ABB RobotStudio station: Step_suction_gripper_20200824-203241.rsstn

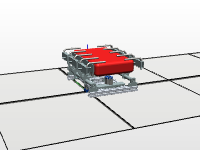
Station Step_suction_gripper (saved by RobotStudio 6.8.8307.1040)
Layout (positions relative to the parent item):
  - T_GRIPPER_2 [graphiccomponentgroup] at (-345.02, -333, 492.44) mm, rotated rx 180 ry 0 rz 0 deg
    - 1046 [graphiccomponentgroup] at (435.5, 105.5, 314.43) mm, rotated rx -90 ry 0 rz 180 deg
      - 1036 [part] at (225.5, -1596.5, -697) mm, rotated rx 0 ry -90 rz -90 deg
      - 1037 [part] at (22.5, 21, 5.41) mm, rotated rx -90 ry 0 rz -90 deg
      - 1038 [part] at (697, -1596.5, 180.5) mm, rotated rx 90 ry 0 rz 180 deg
      - 1039 [part] at (-5.41, 21, -22.5) mm, rotated rx 0 ry 0 rz -90 deg
      - 2.2.001.10.4545.01_kose baglanti duz 45x45_step_MODEL [part]
    - 1048 [graphiccomponentgroup] at (255.5, -60, 272.43) mm, rotated rx 90 ry 0 rz 0 deg
      - 1036 [part] at (225.5, -1596.5, -697) mm, rotated rx 0 ry -90 rz -90 deg
      - 1037 [part] at (22.5, 21, 5.41) mm, rotated rx -90 ry 0 rz -90 deg
      - 1038 [part] at (697, -1596.5, 180.5) mm, rotated rx 90 ry 0 rz 180 deg
      - 1039 [part] at (-5.41, 21, -22.5) mm, rotated rx 0 ry 0 rz -90 deg
      - 2.2.001.10.4545.01_kose baglanti duz 45x45_step_MODEL [part]
    - 1049 [graphiccomponentgroup] at (435.5, 60.5, 272.43) mm, rotated rx 90 ry 0 rz 180 deg
      - 1036 [part] at (225.5, -1596.5, -697) mm, rotated rx 0 ry -90 rz -90 deg
      - 1037 [part] at (22.5, 21, 5.41) mm, rotated rx -90 ry 0 rz -90 deg
      - 1038 [part] at (697, -1596.5, 180.5) mm, rotated rx 90 ry 0 rz 180 deg
      - 1039 [part] at (-5.41, 21, -22.5) mm, rotated rx 0 ry 0 rz -90 deg
      - 2.2.001.10.4545.01_kose baglanti duz 45x45_step_MODEL [part]
    - 1050 [graphiccomponentgroup] at (255.5, 60.5, 314.43) mm, rotated rx -90 ry 0 rz 0 deg
      - 1036 [part] at (225.5, -1596.5, -697) mm, rotated rx 0 ry -90 rz -90 deg
      - 1037 [part] at (22.5, 21, 5.41) mm, rotated rx -90 ry 0 rz -90 deg
      - 1038 [part] at (697, -1596.5, 180.5) mm, rotated rx 90 ry 0 rz 180 deg
      - 1039 [part] at (-5.41, 21, -22.5) mm, rotated rx 0 ry 0 rz -90 deg
      - 2.2.001.10.4545.01_kose baglanti duz 45x45_step_MODEL [part]
    - 1051 [graphiccomponentgroup] at (255, 255, 272.43) mm, rotated rx 90 ry 0 rz -90 deg
      - 1036 [part] at (225.5, -1596.5, -697) mm, rotated rx 0 ry -90 rz -90 deg
      - 1037 [part] at (22.5, 21, 5.41) mm, rotated rx -90 ry 0 rz -90 deg
      - 1038 [part] at (697, -1596.5, 180.5) mm, rotated rx 90 ry 0 rz 180 deg
      - 1039 [part] at (-5.41, 21, -22.5) mm, rotated rx 0 ry 0 rz -90 deg
      - 2.2.001.10.4545.01_kose baglanti duz 45x45_step_MODEL [part]
    - 1052 [graphiccomponentgroup] at (480, -255, 314.43) mm, rotated rx -90 ry 0 rz 90 deg
      - 1036 [part] at (225.5, -1596.5, -697) mm, rotated rx 0 ry -90 rz -90 deg
      - 1037 [part] at (22.5, 21, 5.41) mm, rotated rx -90 ry 0 rz -90 deg
      - 1038 [part] at (697, -1596.5, 180.5) mm, rotated rx 90 ry 0 rz 180 deg
      - 1039 [part] at (-5.41, 21, -22.5) mm, rotated rx 0 ry 0 rz -90 deg
      - 2.2.001.10.4545.01_kose baglanti duz 45x45_step_MODEL [part]
    - 1055 [graphiccomponentgroup] at (255.5, -105, 314.43) mm, rotated rx -90 ry 0 rz 0 deg
      - 1036 [part] at (225.5, -1596.5, -697) mm, rotated rx 0 ry -90 rz -90 deg
      - 1037 [part] at (22.5, 21, 5.41) mm, rotated rx -90 ry 0 rz -90 deg
      - 1038 [part] at (697, -1596.5, 180.5) mm, rotated rx 90 ry 0 rz 180 deg
      - 1039 [part] at (-5.41, 21, -22.5) mm, rotated rx 0 ry 0 rz -90 deg
      - 2.2.001.10.4545.01_kose baglanti duz 45x45_step_MODEL [part]
    - 1059 [graphiccomponentgroup] at (435.5, -105, 272.43) mm, rotated rx 90 ry 0 rz 180 deg
      - 1036 [part] at (225.5, -1596.5, -697) mm, rotated rx 0 ry -90 rz -90 deg
      - 1037 [part] at (22.5, 21, 5.41) mm, rotated rx -90 ry 0 rz -90 deg
      - 1038 [part] at (697, -1596.5, 180.5) mm, rotated rx 90 ry 0 rz 180 deg
      - 1039 [part] at (-5.41, 21, -22.5) mm, rotated rx 0 ry 0 rz -90 deg
      - 2.2.001.10.4545.01_kose baglanti duz 45x45_step_MODEL [part]
    - 1061 [graphiccomponentgroup] at (435, 255, 314.43) mm, rotated rx -90 ry 0 rz -90 deg
      - 1036 [part] at (225.5, -1596.5, -697) mm, rotated rx 0 ry -90 rz -90 deg
      - 1037 [part] at (22.5, 21, 5.41) mm, rotated rx -90 ry 0 rz -90 deg
      - 1038 [part] at (697, -1596.5, 180.5) mm, rotated rx 90 ry 0 rz 180 deg
      - 1039 [part] at (-5.41, 21, -22.5) mm, rotated rx 0 ry 0 rz -90 deg
      - 2.2.001.10.4545.01_kose baglanti duz 45x45_step_MODEL [part]
    - 1062 [graphiccomponentgroup] at (255, -255, 314.43) mm, rotated rx -90 ry 0 rz 90 deg
      - 1036 [part] at (225.5, -1596.5, -697) mm, rotated rx 0 ry -90 rz -90 deg
      - 1037 [part] at (22.5, 21, 5.41) mm, rotated rx -90 ry 0 rz -90 deg
      - 1038 [part] at (697, -1596.5, 180.5) mm, rotated rx 90 ry 0 rz 180 deg
      - 1039 [part] at (-5.41, 21, -22.5) mm, rotated rx 0 ry 0 rz -90 deg
      - 2.2.001.10.4545.01_kose baglanti duz 45x45_step_MODEL [part]
    - 1063 [graphiccomponentgroup] at (537.5, 287.5, 249.93) mm, rotated rx 180 ry 0 rz -90 deg
      - 1035 [graphiccomponentgroup] at (5, 0, 30) mm
        - 1032 [part]
        - 1033 [part]
        - 1034 [part]
      - RULMAN_YATAK [part]
    - 1064 [graphiccomponentgroup] at (435.5, -60, 314.43) mm, rotated rx -90 ry 0 rz 180 deg
      - 1036 [part] at (225.5, -1596.5, -697) mm, rotated rx 0 ry -90 rz -90 deg
      - 1037 [part] at (22.5, 21, 5.41) mm, rotated rx -90 ry 0 rz -90 deg
      - 1038 [part] at (697, -1596.5, 180.5) mm, rotated rx 90 ry 0 rz 180 deg
      - 1039 [part] at (-5.41, 21, -22.5) mm, rotated rx 0 ry 0 rz -90 deg
      - 2.2.001.10.4545.01_kose baglanti duz 45x45_step_MODEL [part]
    - 1065 [graphiccomponentgroup] at (210, 255, 314.43) mm, rotated rx -90 ry 0 rz -90 deg
      - 1036 [part] at (225.5, -1596.5, -697) mm, rotated rx 0 ry -90 rz -90 deg
      - 1037 [part] at (22.5, 21, 5.41) mm, rotated rx -90 ry 0 rz -90 deg
      - 1038 [part] at (697, -1596.5, 180.5) mm, rotated rx 90 ry 0 rz 180 deg
      - 1039 [part] at (-5.41, 21, -22.5) mm, rotated rx 0 ry 0 rz -90 deg
      - 2.2.001.10.4545.01_kose baglanti duz 45x45_step_MODEL [part]
    - 1066 [graphiccomponentgroup] at (255.5, 105.5, 272.43) mm, rotated rx 90 ry 0 rz 0 deg
      - 1036 [part] at (225.5, -1596.5, -697) mm, rotated rx 0 ry -90 rz -90 deg
      - 1037 [part] at (22.5, 21, 5.41) mm, rotated rx -90 ry 0 rz -90 deg
      - 1038 [part] at (697, -1596.5, 180.5) mm, rotated rx 90 ry 0 rz 180 deg
      - 1039 [part] at (-5.41, 21, -22.5) mm, rotated rx 0 ry 0 rz -90 deg
      - 2.2.001.10.4545.01_kose baglanti duz 45x45_step_MODEL [part]
    - 1067 [graphiccomponentgroup] at (152.5, -287.5, 249.93) mm, rotated rx 180 ry 0 rz 90 deg
      - 1035 [graphiccomponentgroup] at (5, 0, 30) mm
        - 1032 [part]
        - 1033 [part]
        - 1034 [part]
      - RULMAN_YATAK [part]
    - 1070 [graphiccomponentgroup] at (538.22, -287.5, 251.07) mm, rotated rx 180 ry 0 rz 90 deg
      - 1035 [graphiccomponentgroup] at (5, 0, 30) mm
        - 1032 [part]
        - 1033 [part]
        - 1034 [part]
      - RULMAN_YATAK [part]
    - 1071 [graphiccomponentgroup] at (152.5, 287.5, 249.93) mm, rotated rx 180 ry 0 rz -90 deg
      - 1035 [graphiccomponentgroup] at (5, 0, 30) mm
        - 1032 [part]
        - 1033 [part]
        - 1034 [part]
      - RULMAN_YATAK [part]
    - 1072 [graphiccomponentgroup] at (435, -255, 272.43) mm, rotated rx 90 ry 0 rz 90 deg
      - 1036 [part] at (225.5, -1596.5, -697) mm, rotated rx 0 ry -90 rz -90 deg
      - 1037 [part] at (22.5, 21, 5.41) mm, rotated rx -90 ry 0 rz -90 deg
      - 1038 [part] at (697, -1596.5, 180.5) mm, rotated rx 90 ry 0 rz 180 deg
      - 1039 [part] at (-5.41, 21, -22.5) mm, rotated rx 0 ry 0 rz -90 deg
      - 2.2.001.10.4545.01_kose baglanti duz 45x45_step_MODEL [part]
    - 1073 [graphiccomponentgroup] at (480, 255, 272.43) mm, rotated rx 90 ry 0 rz -90 deg
      - 1036 [part] at (225.5, -1596.5, -697) mm, rotated rx 0 ry -90 rz -90 deg
      - 1037 [part] at (22.5, 21, 5.41) mm, rotated rx -90 ry 0 rz -90 deg
      - 1038 [part] at (697, -1596.5, 180.5) mm, rotated rx 90 ry 0 rz 180 deg
      - 1039 [part] at (-5.41, 21, -22.5) mm, rotated rx 0 ry 0 rz -90 deg
      - 2.2.001.10.4545.01_kose baglanti duz 45x45_step_MODEL [part]
    - 1075 [graphiccomponentgroup] at (210, -255, 272.43) mm, rotated rx 90 ry 0 rz 90 deg
      - 1036 [part] at (225.5, -1596.5, -697) mm, rotated rx 0 ry -90 rz -90 deg
      - 1037 [part] at (22.5, 21, 5.41) mm, rotated rx -90 ry 0 rz -90 deg
      - 1038 [part] at (697, -1596.5, 180.5) mm, rotated rx 90 ry 0 rz 180 deg
      - 1039 [part] at (-5.41, 21, -22.5) mm, rotated rx 0 ry 0 rz -90 deg
      - 2.2.001.10.4545.01_kose baglanti duz 45x45_step_MODEL [part]
    - 1076 [graphiccomponentgroup] at (152.5, -244, 219.93) mm, rotated rx -1.14 ry 0 rz 90 deg
      - 1021 [graphiccomponentgroup] at (505.5, 0, 0) mm, rotated rx 180 ry 0 rz 180 deg
        - 1005 [part] at (523, 0, 0) mm, rotated rx 0 ry 0 rz -90 deg
        - 1006 [part] at (0, 0, 0) mm, rotated rx 0 ry 0 rz 90 deg
        - GR1_P1-2 [part]
      - 1022 [graphiccomponentgroup] at (244, -1, -144) mm, rotated rx 0 ry 90 rz -90 deg
        - 1007 [part] at (0, 215, 0.5) mm, rotated rx -90 ry 0 rz 180 deg
        - 1008 [part] at (0, -35, 0.5) mm, rotated rx -90 ry 0 rz 180 deg
        - 1009 [part] at (0, -215, 0.5) mm, rotated rx -90 ry 0 rz 180 deg
        - GR1_P4 [part]
      - 1023 [part] at (371.5, 54.54, -79.76) mm, rotated rx 0 ry 0.38 rz -90 deg
      - 1024 [part] at (394, 68.87, -207.14) mm, rotated rx 0 ry 0.38 rz -90 deg
      - 1025 [part] at (244, 68.47, -146.98) mm, rotated rx 0.38 ry 0 rz 0 deg
      - 1026 [part] at (94, 68.87, -207.14) mm, rotated rx 0 ry 0.38 rz -90 deg
      - 1027 [part] at (-56, 68.87, -207.14) mm, rotated rx 0 ry 0.38 rz -90 deg
      - 1028 [part] at (244, 68.87, -207.14) mm, rotated rx 0 ry 0.38 rz -90 deg
      - 1029 [part] at (124.5, 54.54, -79.76) mm, rotated rx 0 ry 0.38 rz -90 deg
      - 1030 [part] at (544, 68.87, -207.14) mm, rotated rx 0 ry 0.38 rz -90 deg
      - 1031 [part] at (-94, 0, 0) mm, rotated rx 0 ry 30.38 rz 90 deg
    - 1077 [graphiccomponentgroup] at (538.22, 244, 221.07) mm, rotated rx -0.38 ry 0 rz -90 deg
      - 1010 [graphiccomponentgroup] at (-17.5, 0, 0) mm
        - 1005 [part] at (523, 0, 0) mm, rotated rx 0 ry 0 rz -90 deg
        - 1006 [part] at (0, 0, 0) mm, rotated rx 0 ry 0 rz 90 deg
        - GR1_P1-2 [part]
      - 1011 [graphiccomponentgroup] at (244, -1, -144) mm, rotated rx 0 ry 90 rz -90 deg
        - 1007 [part] at (0, 215, 0.5) mm, rotated rx -90 ry 0 rz 180 deg
        - 1008 [part] at (0, -35, 0.5) mm, rotated rx -90 ry 0 rz 180 deg
        - 1009 [part] at (0, -215, 0.5) mm, rotated rx -90 ry 0 rz 180 deg
        - GR1_P4 [part]
      - 1012 [part] at (371.5, 54.54, -79.76) mm, rotated rx 0 ry 0.38 rz -90 deg
      - 1013 [part] at (394, 68.87, -207.14) mm, rotated rx 0 ry 0.38 rz -90 deg
      - 1014 [part] at (244, 68.47, -146.98) mm, rotated rx 0.38 ry 0 rz 0 deg
      - 1015 [part] at (94, 68.87, -207.14) mm, rotated rx 0 ry 0.38 rz -90 deg
      - 1016 [part] at (-56, 68.87, -207.14) mm, rotated rx 0 ry 0.38 rz -90 deg
      - 1017 [part] at (244, 68.87, -207.14) mm, rotated rx 0 ry 0.38 rz -90 deg
      - 1018 [part] at (124.5, 54.54, -79.76) mm, rotated rx 0 ry 0.38 rz -90 deg
      - 1019 [part] at (544, 68.87, -207.14) mm, rotated rx 0 ry 0.38 rz -90 deg
      - 1020 [part] at (572, 0, 0) mm, rotated rx 0 ry 30.38 rz 90 deg
    - 1079 [graphiccomponentgroup] at (345.02, -333, 408.94) mm, rotated rx 180 ry 0 rz 180 deg
      - 1003 [part]
      - 1004 [part]
    - 1084 [graphiccomponentgroup] at (345, -179.5, 242.67) mm, rotated rx 180 ry 0 rz 90 deg
      - 1001 [part] at (0, 0, 33) mm
      - 1002 [part]
    - 1085 [graphiccomponentgroup] at (345, 179.5, 242.67) mm, rotated rx 180 ry 0 rz -90 deg
      - 1001 [part] at (0, 0, 33) mm
      - 1002 [part]
    - 1047 [part] at (375, -82.5, 294.93) mm, rotated rx 0 ry -90 rz -180 deg
    - 1053 [part] at (375, 82.5, 294.93) mm, rotated rx 0 ry -90 rz -180 deg
    - 1054 [part] at (-110, 277.5, 294.93) mm, rotated rx 0 ry -90 rz -180 deg
    - CAJA [part] at (-1373.11, 0, 0) mm
    - 1057 [part] at (345, -2.5, 317.43) mm
    - 1058 [part] at (-110, -277.5, 294.93) mm, rotated rx 0 ry -90 rz -180 deg
    - 1060 [part] at (232.5, -480, 294.93) mm, rotated rx 0 ry -90 rz -90 deg
    - 1069 [part] at (457.5, -480, 294.93) mm, rotated rx 0 ry -90 rz -90 deg
    - 1078 [part] at (265.02, -345.5, 237.16) mm, rotated rx 0 ry 0 rz 90 deg
    - 1080 [part] at (345.02, -300, 317.44) mm, rotated rx 0 ry 0 rz 90 deg
    - 1081 [part] at (345, 0, 147.17) mm, rotated rx 180 ry 0 rz 180 deg
    - 1082 [part] at (345, -182, 257.67) mm, rotated rx 0 ry 0 rz 90 deg
    - 1083 [part] at (345, 248, 251.67) mm, rotated rx 0 ry 0 rz 90 deg
    - 1086 [part] at (345, -149.5, 295.17) mm, rotated rx 0 ry 0 rz -90 deg
    - 1087 [part] at (345, 150.5, 295.17) mm, rotated rx 0 ry 0 rz 90 deg
